// TIA Portal V20 export
TYPE "LKinCtrl_typeCmdLoggerElement"
   STRUCT
      cmdType : Int := -1;   // 1: MoveLinAbs; 2: MoveLinRel; 3: MoveCircAbs; 4: MoveCircRel; 5: MoveDirectAbs; 6: MoveDirectRel; 10: TrackConveyorBelt; 100: WaitTime; 40/41/42: ContourOffset; 0: FlagOnlyCmd; -1: End of List
      pathDataName : String["LKINCTRL_LENGTH_OF_PATHDATA_NAME"];   // name of PathData
      pathDataIdentifier : Int;   // identifier of PathData containing command
      cmdID : DInt;   // to be set to PathDataOperate[list position] by PreBuffer for identification in ExecuteBuffer
      cmdName : String[4];   // command name
      coordinateX : LReal;   // X (linear) / endPoint[1] (circular)
      coordinateY : LReal;   // Y (linear) / endPoint[2] (circular)
      coordinateZ : LReal;   // Z (linear) / endPoint[3] (circular)
      coordinateA : LReal;   // A (linear) / endPoint[4] (circular)
      coordSystem : DInt := 0;   // 0: WCS; 1: OCS[1]; 2: OCS[2]; 3: OCS[3]
      bufferMode : DInt := 1;   // 1: standstill between commands, 2: blending with lower speed; 5: blending with higher speed
      transitionParameter : LReal;   // blending distance - >0.0: configured value used; <0.0: maximum possible blending distance used
      dynVelocity : LReal;   // >0.0: configured value used; <0.0: default TO setting used
      dynAcceleration : LReal;   // >0.0: configured value used; <0.0: default TO setting used
      dynDeceleration : LReal;   // >0.0: configured value used; <0.0: default TO setting used
      dynJerk : LReal;   // >0.0: configured value used; <0.0: default TO setting used
      dynamicAdpation : DInt;   // <0.0: default TO setting used; 0: no dynamic adaption; 1: with variable limits; 2: with constant limits
      linkConstellation : DWord;   // linkConstellation (effective for MoveDirect commands only)
      positionMode : DInt;   // 1: absolute cartesian position and absolute orientation; 2: absolute cartesian position and relative orientation (effective for MoveDirect commands only)
      circMode : DInt;   // 0: auxPoint defines point on circle line; 1: auxPoint defines circle center; 2: radius and endPoint define circle segment
      auxPoint_1 : LReal;   // auxiliary point for circle definition
      auxPoint_2 : LReal;   // auxiliary point for circle definition
      auxPoint_3 : LReal;   // auxiliary point for circle definition
      pathChoice : DInt;   // circMode(0): not relevant; circMode(1): 0: pos direction; 1: neg direction; circMode(2): 0: short pos segment; 1: short neg segment; 2: long pos segment; 3: long neg segment
      circlePlane : DInt;   // circMode(0): not relevant; circMode(1+2): 0: XZ; 1: YZ; 2: XY
      radius : LReal;   // only in combination with circMode(2): radius
      arc : LReal;   // only in combination with circMode(1): arc
   END_STRUCT;
END_TYPE
